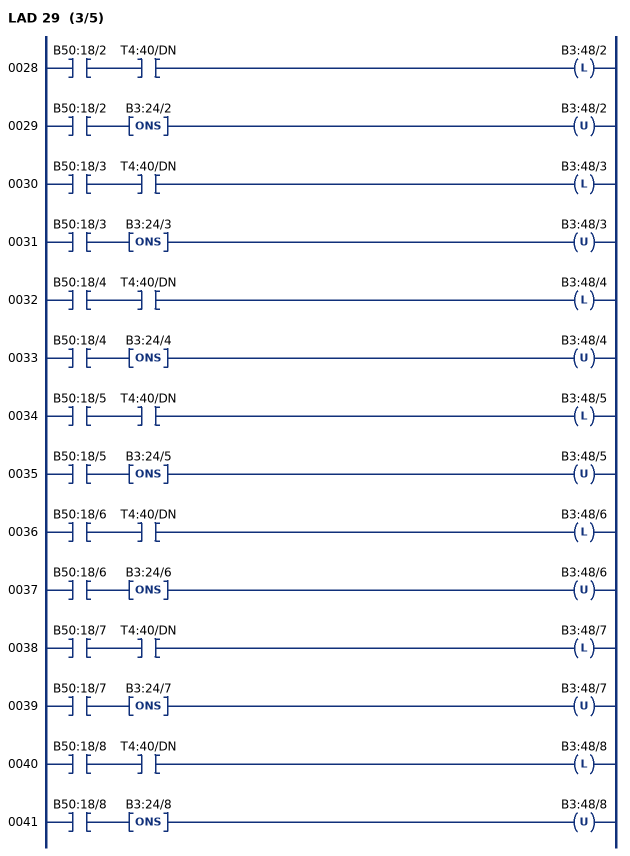
% Rung: 28 %
SOR XIC B50:18/2 XIC T4:40/DN OTL B3:48/2 EOR
% Rung: 29 %
SOR XIC B50:18/2 OSR B3:24/2 OTU B3:48/2 EOR
% Rung: 30 %
SOR XIC B50:18/3 XIC T4:40/DN OTL B3:48/3 EOR
% Rung: 31 %
SOR XIC B50:18/3 OSR B3:24/3 OTU B3:48/3 EOR
% Rung: 32 %
SOR XIC B50:18/4 XIC T4:40/DN OTL B3:48/4 EOR
% Rung: 33 %
SOR XIC B50:18/4 OSR B3:24/4 OTU B3:48/4 EOR
% Rung: 34 %
SOR XIC B50:18/5 XIC T4:40/DN OTL B3:48/5 EOR
% Rung: 35 %
SOR XIC B50:18/5 OSR B3:24/5 OTU B3:48/5 EOR
% Rung: 36 %
SOR XIC B50:18/6 XIC T4:40/DN OTL B3:48/6 EOR
% Rung: 37 %
SOR XIC B50:18/6 OSR B3:24/6 OTU B3:48/6 EOR
% Rung: 38 %
SOR XIC B50:18/7 XIC T4:40/DN OTL B3:48/7 EOR
% Rung: 39 %
SOR XIC B50:18/7 OSR B3:24/7 OTU B3:48/7 EOR
% Rung: 40 %
SOR XIC B50:18/8 XIC T4:40/DN OTL B3:48/8 EOR
% Rung: 41 %
SOR XIC B50:18/8 OSR B3:24/8 OTU B3:48/8 EOR

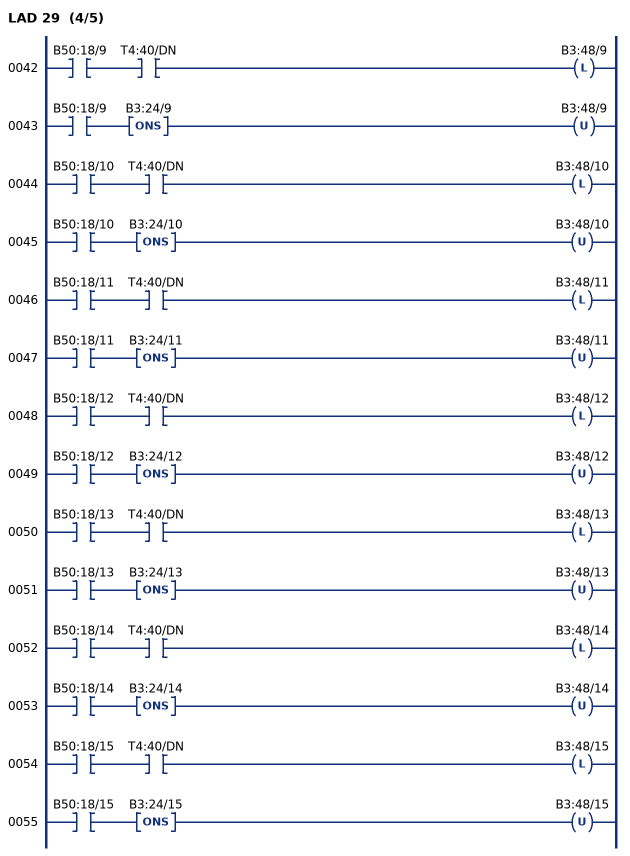
% Rung: 42 %
SOR XIC B50:18/9 XIC T4:40/DN OTL B3:48/9 EOR
% Rung: 43 %
SOR XIC B50:18/9 OSR B3:24/9 OTU B3:48/9 EOR
% Rung: 44 %
SOR XIC B50:18/10 XIC T4:40/DN OTL B3:48/10 EOR
% Rung: 45 %
SOR XIC B50:18/10 OSR B3:24/10 OTU B3:48/10 EOR
% Rung: 46 %
SOR XIC B50:18/11 XIC T4:40/DN OTL B3:48/11 EOR
% Rung: 47 %
SOR XIC B50:18/11 OSR B3:24/11 OTU B3:48/11 EOR
% Rung: 48 %
SOR XIC B50:18/12 XIC T4:40/DN OTL B3:48/12 EOR
% Rung: 49 %
SOR XIC B50:18/12 OSR B3:24/12 OTU B3:48/12 EOR
% Rung: 50 %
SOR XIC B50:18/13 XIC T4:40/DN OTL B3:48/13 EOR
% Rung: 51 %
SOR XIC B50:18/13 OSR B3:24/13 OTU B3:48/13 EOR
% Rung: 52 %
SOR XIC B50:18/14 XIC T4:40/DN OTL B3:48/14 EOR
% Rung: 53 %
SOR XIC B50:18/14 OSR B3:24/14 OTU B3:48/14 EOR
% Rung: 54 %
SOR XIC B50:18/15 XIC T4:40/DN OTL B3:48/15 EOR
% Rung: 55 %
SOR XIC B50:18/15 OSR B3:24/15 OTU B3:48/15 EOR

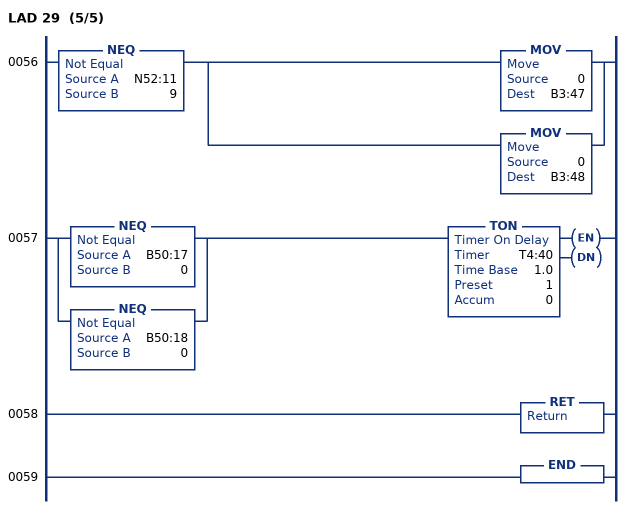
% Rung: 56 %
SOR NEQ N52:11 9 BST MOV 0 B3:47 NXB MOV 0 B3:48 BND EOR
% Rung: 57 %
SOR BST NEQ B50:17 0 NXB NEQ B50:18 0 BND TON T4:40 1.0 1 0 EOR
% Rung: 58 %
SOR RET EOR
% Rung: 59 %
SOR END EOR

LADDER 30
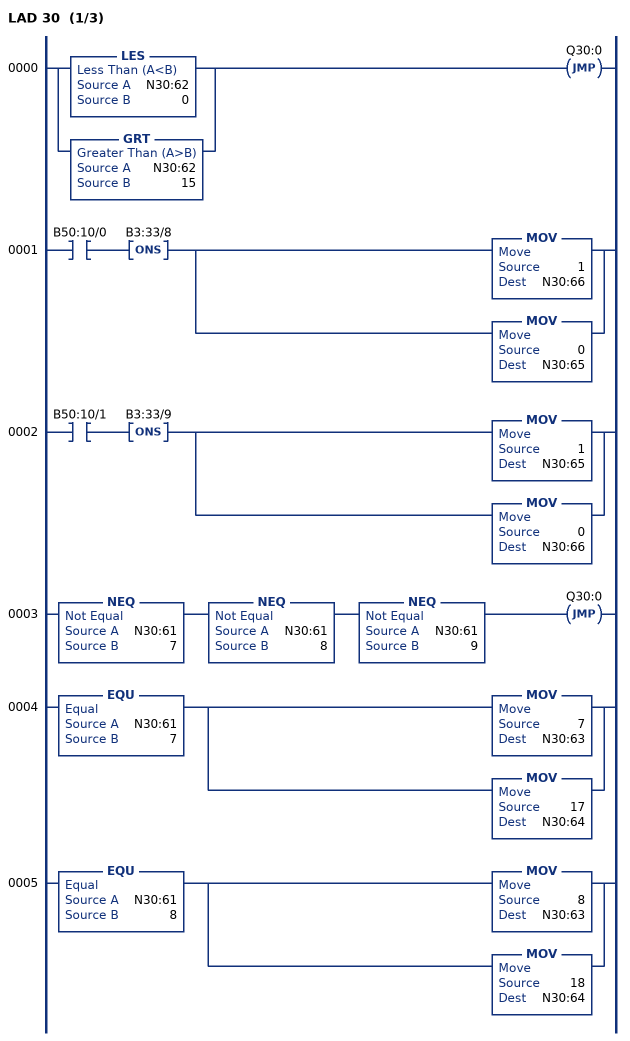
% Rung: 0 %
SOR BST LES N30:62 0 NXB GRT N30:62 15 BND JMP Q30:0 EOR
% Rung: 1 %
SOR XIC B50:10/0 OSR B3:33/8 BST MOV 1 N30:66 NXB MOV 0 N30:65 BND EOR
% Rung: 2 %
SOR XIC B50:10/1 OSR B3:33/9 BST MOV 1 N30:65 NXB MOV 0 N30:66 BND EOR
% Rung: 3 %
SOR NEQ N30:61 7 NEQ N30:61 8 NEQ N30:61 9 JMP Q30:0 EOR
% Rung: 4 %
SOR EQU N30:61 7 BST MOV 7 N30:63 NXB MOV 17 N30:64 BND EOR
% Rung: 5 %
SOR EQU N30:61 8 BST MOV 8 N30:63 NXB MOV 18 N30:64 BND EOR

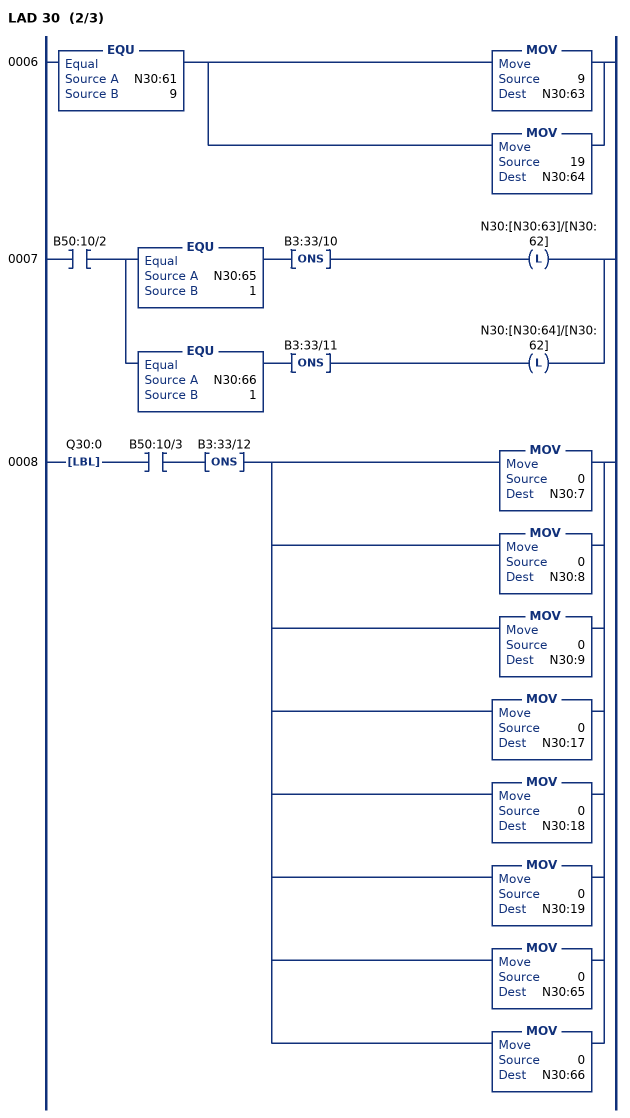
% Rung: 6 %
SOR EQU N30:61 9 BST MOV 9 N30:63 NXB MOV 19 N30:64 BND EOR
% Rung: 7 %
SOR XIC B50:10/2 BST EQU N30:65 1 OSR B3:33/10 OTL N30:[N30:63]/[N30:62] NXB EQU N30:66 1 OSR B3:33/11 OTL N30:[N30:64]/[N30:62] BND EOR
% Rung: 8 %
SOR LBL Q30:0 XIC B50:10/3 OSR B3:33/12 BST MOV 0 N30:7 NXB MOV 0 N30:8 NXB MOV 0 N30:9 NXB MOV 0 N30:17 NXB MOV 0 N30:18 NXB MOV 0 N30:19 NXB MOV 0 N30:65 NXB MOV 0 N30:66 BND EOR

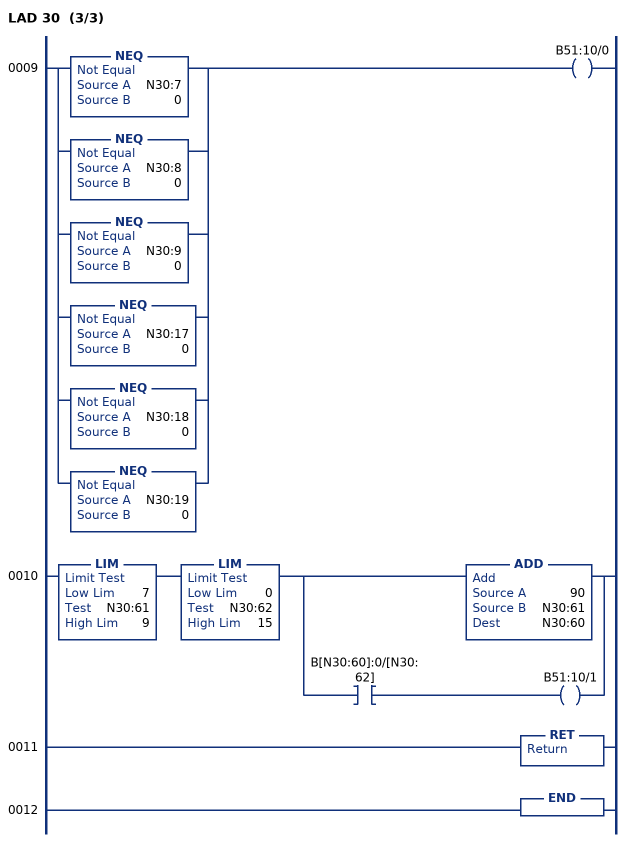
% Rung: 9 %
SOR BST NEQ N30:7 0 NXB NEQ N30:8 0 NXB NEQ N30:9 0 NXB NEQ N30:17 0 NXB NEQ N30:18 0 NXB NEQ N30:19 0 BND OTE B51:10/0 EOR
% Rung: 10 %
SOR LIM 7 N30:61 9 LIM 0 N30:62 15 BST ADD 90 N30:61 N30:60 NXB XIC B[N30:60]:0/[N30:62] OTE B51:10/1 BND EOR
% Rung: 11 %
SOR RET EOR
% Rung: 12 %
SOR END EOR

LADDER 31
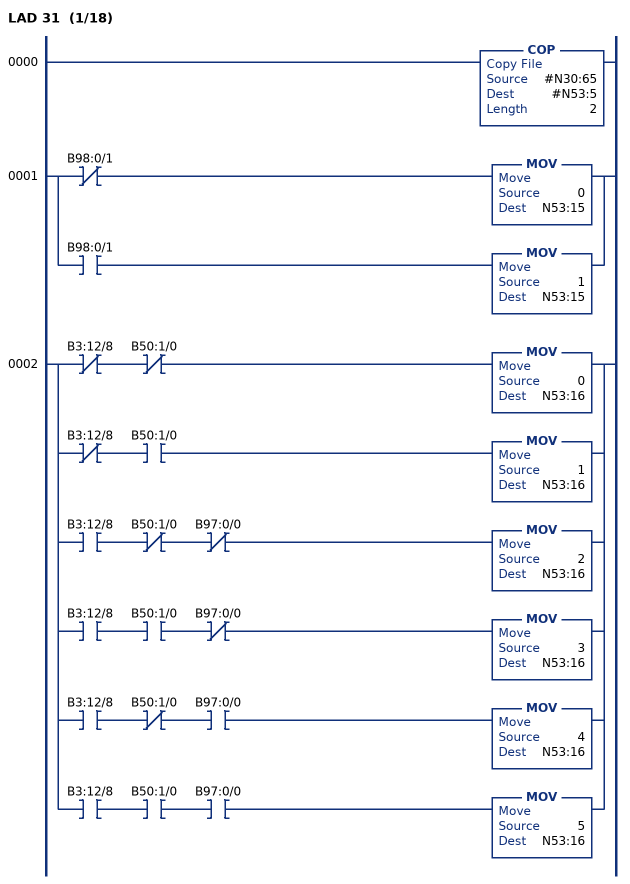
% Rung: 0 %
SOR COP #N30:65 #N53:5 2 EOR
% Rung: 1 %
SOR BST XIO B98:0/1 MOV 0 N53:15 NXB XIC B98:0/1 MOV 1 N53:15 BND EOR
% Rung: 2 %
SOR BST XIO B3:12/8 XIO B50:1/0 MOV 0 N53:16 NXB XIO B3:12/8 XIC B50:1/0 MOV 1 N53:16 NXB XIC B3:12/8 XIO B50:1/0 XIO B97:0/0 MOV 2 N53:16 NXB XIC B3:12/8 XIC B50:1/0 XIO B97:0/0 MOV 3 N53:16 NXB XIC B3:12/8 XIO B50:1/0 XIC B97:0/0 MOV 4 N53:16 NXB XIC B3:12/8 XIC B50:1/0 XIC B97:0/0 MOV 5 N53:16 BND EOR

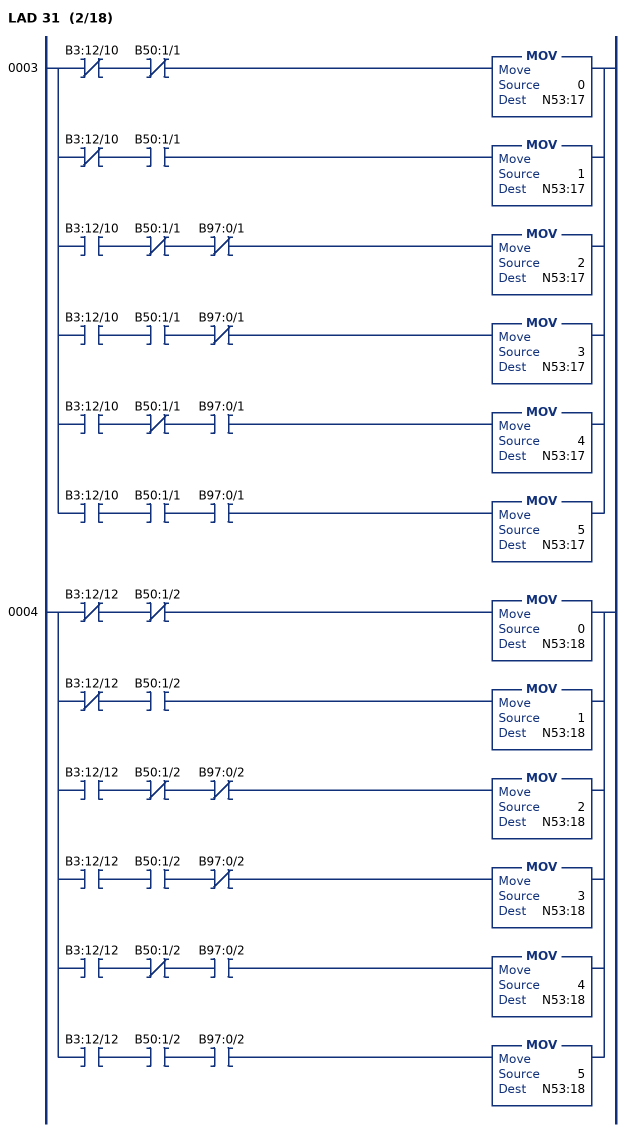
% Rung: 3 %
SOR BST XIO B3:12/10 XIO B50:1/1 MOV 0 N53:17 NXB XIO B3:12/10 XIC B50:1/1 MOV 1 N53:17 NXB XIC B3:12/10 XIO B50:1/1 XIO B97:0/1 MOV 2 N53:17 NXB XIC B3:12/10 XIC B50:1/1 XIO B97:0/1 MOV 3 N53:17 NXB XIC B3:12/10 XIO B50:1/1 XIC B97:0/1 MOV 4 N53:17 NXB XIC B3:12/10 XIC B50:1/1 XIC B97:0/1 MOV 5 N53:17 BND EOR
% Rung: 4 %
SOR BST XIO B3:12/12 XIO B50:1/2 MOV 0 N53:18 NXB XIO B3:12/12 XIC B50:1/2 MOV 1 N53:18 NXB XIC B3:12/12 XIO B50:1/2 XIO B97:0/2 MOV 2 N53:18 NXB XIC B3:12/12 XIC B50:1/2 XIO B97:0/2 MOV 3 N53:18 NXB XIC B3:12/12 XIO B50:1/2 XIC B97:0/2 MOV 4 N53:18 NXB XIC B3:12/12 XIC B50:1/2 XIC B97:0/2 MOV 5 N53:18 BND EOR

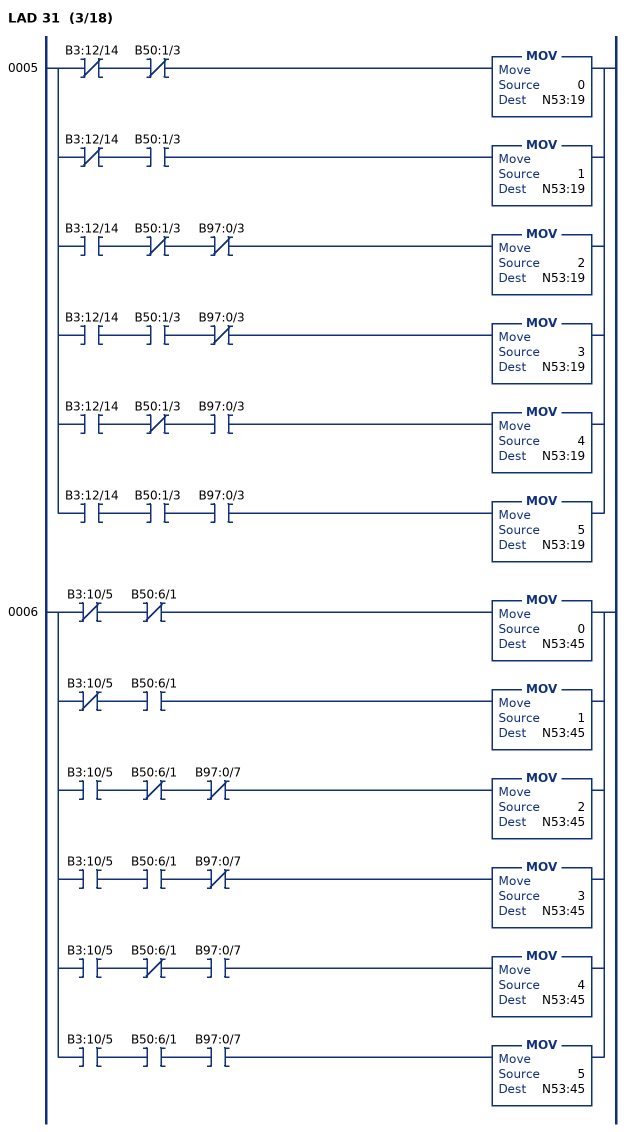
% Rung: 5 %
SOR BST XIO B3:12/14 XIO B50:1/3 MOV 0 N53:19 NXB XIO B3:12/14 XIC B50:1/3 MOV 1 N53:19 NXB XIC B3:12/14 XIO B50:1/3 XIO B97:0/3 MOV 2 N53:19 NXB XIC B3:12/14 XIC B50:1/3 XIO B97:0/3 MOV 3 N53:19 NXB XIC B3:12/14 XIO B50:1/3 XIC B97:0/3 MOV 4 N53:19 NXB XIC B3:12/14 XIC B50:1/3 XIC B97:0/3 MOV 5 N53:19 BND EOR
% Rung: 6 %
SOR BST XIO B3:10/5 XIO B50:6/1 MOV 0 N53:45 NXB XIO B3:10/5 XIC B50:6/1 MOV 1 N53:45 NXB XIC B3:10/5 XIO B50:6/1 XIO B97:0/7 MOV 2 N53:45 NXB XIC B3:10/5 XIC B50:6/1 XIO B97:0/7 MOV 3 N53:45 NXB XIC B3:10/5 XIO B50:6/1 XIC B97:0/7 MOV 4 N53:45 NXB XIC B3:10/5 XIC B50:6/1 XIC B97:0/7 MOV 5 N53:45 BND EOR

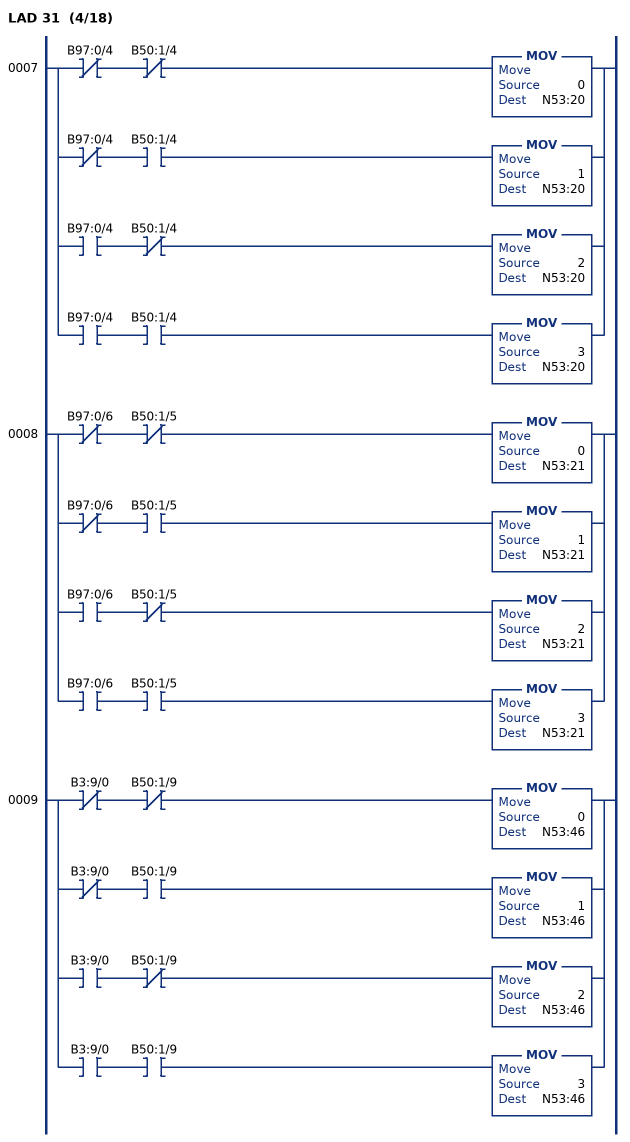
% Rung: 7 %
SOR BST XIO B97:0/4 XIO B50:1/4 MOV 0 N53:20 NXB XIO B97:0/4 XIC B50:1/4 MOV 1 N53:20 NXB XIC B97:0/4 XIO B50:1/4 MOV 2 N53:20 NXB XIC B97:0/4 XIC B50:1/4 MOV 3 N53:20 BND EOR
% Rung: 8 %
SOR BST XIO B97:0/6 XIO B50:1/5 MOV 0 N53:21 NXB XIO B97:0/6 XIC B50:1/5 MOV 1 N53:21 NXB XIC B97:0/6 XIO B50:1/5 MOV 2 N53:21 NXB XIC B97:0/6 XIC B50:1/5 MOV 3 N53:21 BND EOR
% Rung: 9 %
SOR BST XIO B3:9/0 XIO B50:1/9 MOV 0 N53:46 NXB XIO B3:9/0 XIC B50:1/9 MOV 1 N53:46 NXB XIC B3:9/0 XIO B50:1/9 MOV 2 N53:46 NXB XIC B3:9/0 XIC B50:1/9 MOV 3 N53:46 BND EOR

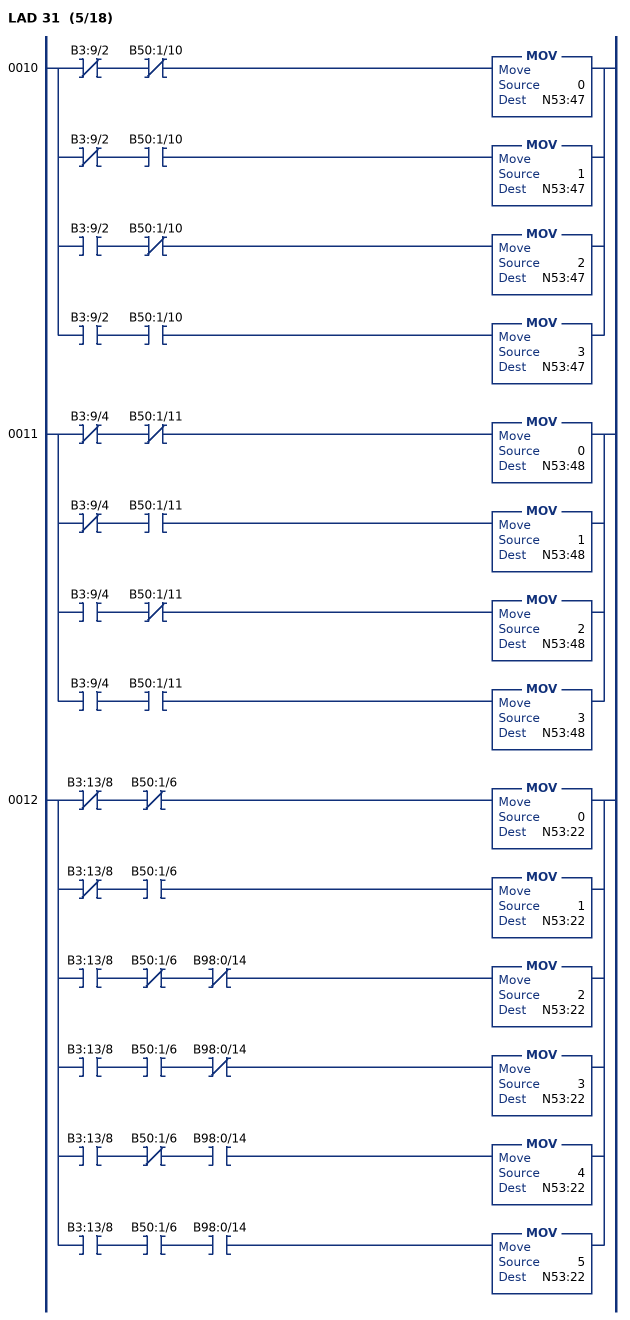
% Rung: 10 %
SOR BST XIO B3:9/2 XIO B50:1/10 MOV 0 N53:47 NXB XIO B3:9/2 XIC B50:1/10 MOV 1 N53:47 NXB XIC B3:9/2 XIO B50:1/10 MOV 2 N53:47 NXB XIC B3:9/2 XIC B50:1/10 MOV 3 N53:47 BND EOR
% Rung: 11 %
SOR BST XIO B3:9/4 XIO B50:1/11 MOV 0 N53:48 NXB XIO B3:9/4 XIC B50:1/11 MOV 1 N53:48 NXB XIC B3:9/4 XIO B50:1/11 MOV 2 N53:48 NXB XIC B3:9/4 XIC B50:1/11 MOV 3 N53:48 BND EOR
% Rung: 12 %
SOR BST XIO B3:13/8 XIO B50:1/6 MOV 0 N53:22 NXB XIO B3:13/8 XIC B50:1/6 MOV 1 N53:22 NXB XIC B3:13/8 XIO B50:1/6 XIO B98:0/14 MOV 2 N53:22 NXB XIC B3:13/8 XIC B50:1/6 XIO B98:0/14 MOV 3 N53:22 NXB XIC B3:13/8 XIO B50:1/6 XIC B98:0/14 MOV 4 N53:22 NXB XIC B3:13/8 XIC B50:1/6 XIC B98:0/14 MOV 5 N53:22 BND EOR

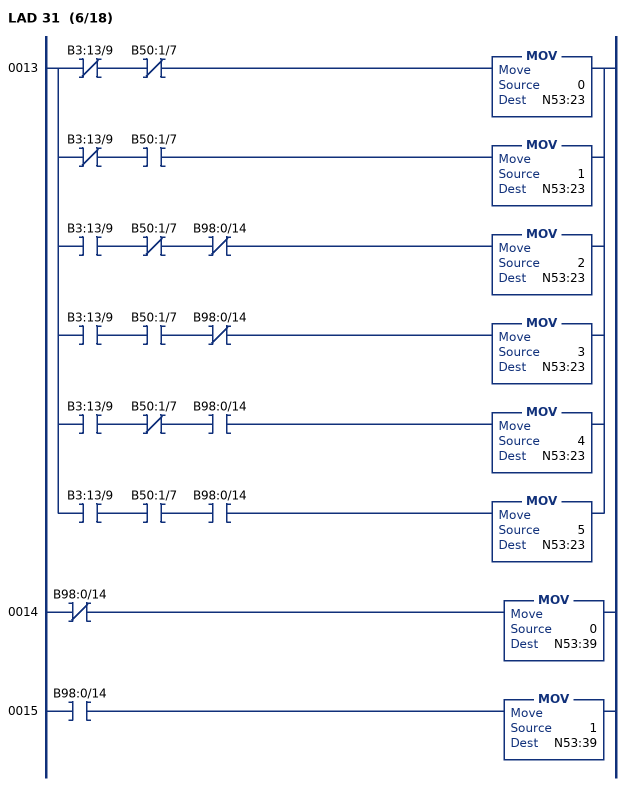
% Rung: 13 %
SOR BST XIO B3:13/9 XIO B50:1/7 MOV 0 N53:23 NXB XIO B3:13/9 XIC B50:1/7 MOV 1 N53:23 NXB XIC B3:13/9 XIO B50:1/7 XIO B98:0/14 MOV 2 N53:23 NXB XIC B3:13/9 XIC B50:1/7 XIO B98:0/14 MOV 3 N53:23 NXB XIC B3:13/9 XIO B50:1/7 XIC B98:0/14 MOV 4 N53:23 NXB XIC B3:13/9 XIC B50:1/7 XIC B98:0/14 MOV 5 N53:23 BND EOR
% Rung: 14 %
SOR XIO B98:0/14 MOV 0 N53:39 EOR
% Rung: 15 %
SOR XIC B98:0/14 MOV 1 N53:39 EOR

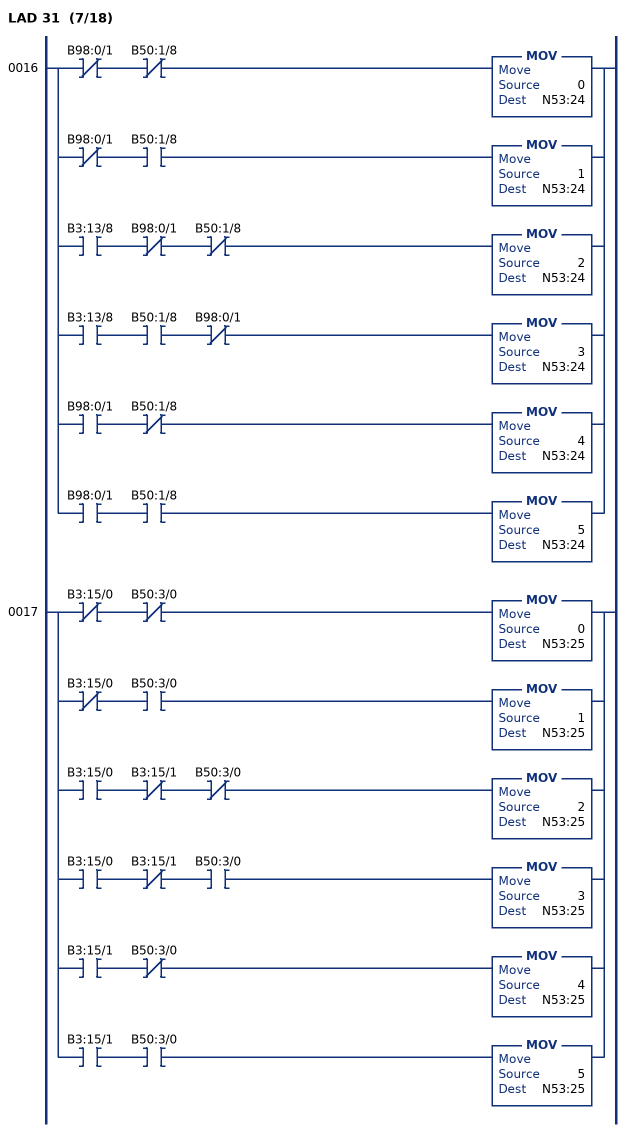
% Rung: 16 %
SOR BST XIO B98:0/1 XIO B50:1/8 MOV 0 N53:24 NXB XIO B98:0/1 XIC B50:1/8 MOV 1 N53:24 NXB XIC B3:13/8 XIO B98:0/1 XIO B50:1/8 MOV 2 N53:24 NXB XIC B3:13/8 XIC B50:1/8 XIO B98:0/1 MOV 3 N53:24 NXB XIC B98:0/1 XIO B50:1/8 MOV 4 N53:24 NXB XIC B98:0/1 XIC B50:1/8 MOV 5 N53:24 BND EOR
% Rung: 17 %
SOR BST XIO B3:15/0 XIO B50:3/0 MOV 0 N53:25 NXB XIO B3:15/0 XIC B50:3/0 MOV 1 N53:25 NXB XIC B3:15/0 XIO B3:15/1 XIO B50:3/0 MOV 2 N53:25 NXB XIC B3:15/0 XIO B3:15/1 XIC B50:3/0 MOV 3 N53:25 NXB XIC B3:15/1 XIO B50:3/0 MOV 4 N53:25 NXB XIC B3:15/1 XIC B50:3/0 MOV 5 N53:25 BND EOR

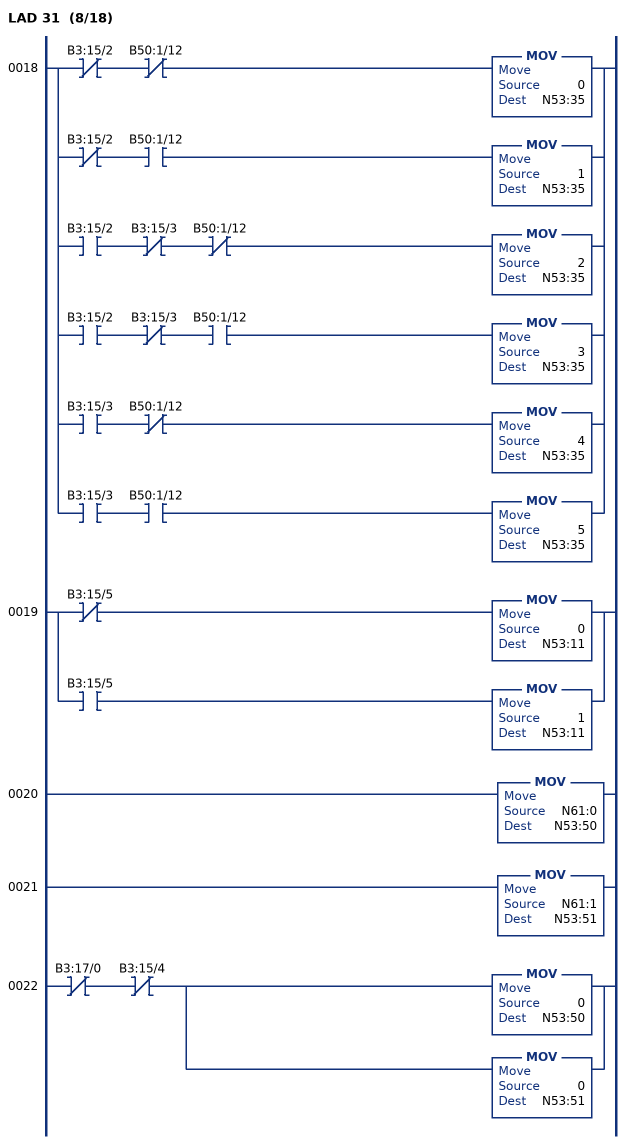
% Rung: 18 %
SOR BST XIO B3:15/2 XIO B50:1/12 MOV 0 N53:35 NXB XIO B3:15/2 XIC B50:1/12 MOV 1 N53:35 NXB XIC B3:15/2 XIO B3:15/3 XIO B50:1/12 MOV 2 N53:35 NXB XIC B3:15/2 XIO B3:15/3 XIC B50:1/12 MOV 3 N53:35 NXB XIC B3:15/3 XIO B50:1/12 MOV 4 N53:35 NXB XIC B3:15/3 XIC B50:1/12 MOV 5 N53:35 BND EOR
% Rung: 19 %
SOR BST XIO B3:15/5 MOV 0 N53:11 NXB XIC B3:15/5 MOV 1 N53:11 BND EOR
% Rung: 20 %
SOR MOV N61:0 N53:50 EOR
% Rung: 21 %
SOR MOV N61:1 N53:51 EOR
% Rung: 22 %
SOR XIO B3:17/0 XIO B3:15/4 BST MOV 0 N53:50 NXB MOV 0 N53:51 BND EOR

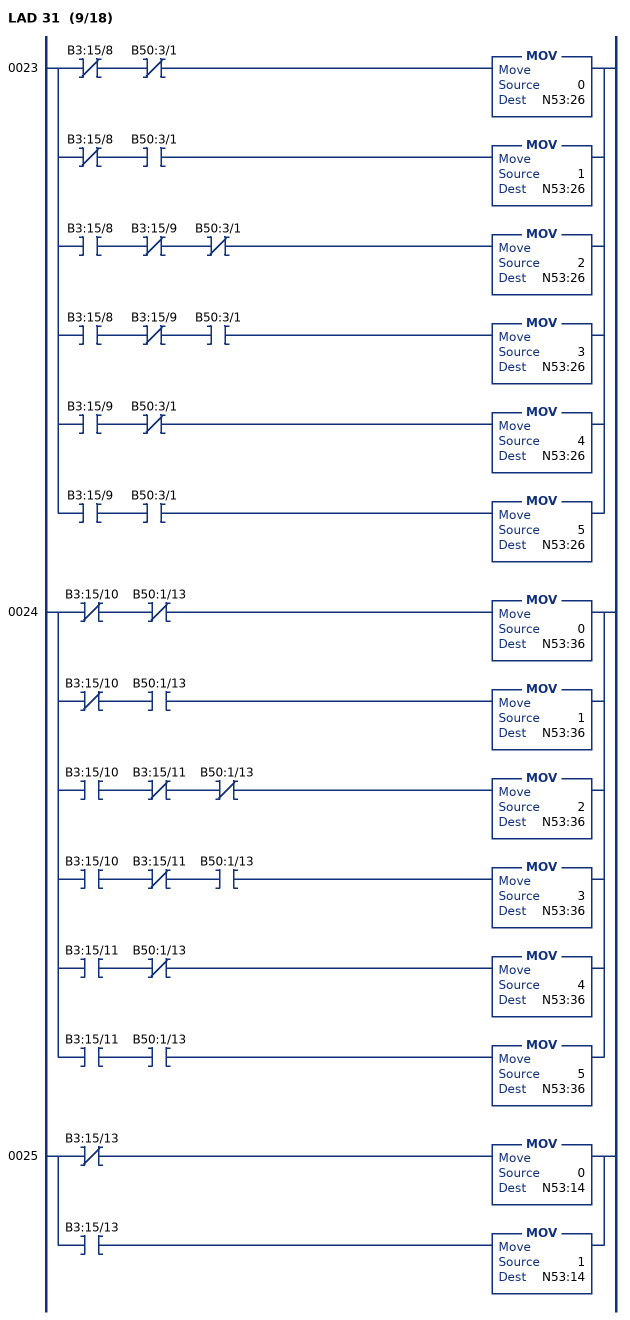
% Rung: 23 %
SOR BST XIO B3:15/8 XIO B50:3/1 MOV 0 N53:26 NXB XIO B3:15/8 XIC B50:3/1 MOV 1 N53:26 NXB XIC B3:15/8 XIO B3:15/9 XIO B50:3/1 MOV 2 N53:26 NXB XIC B3:15/8 XIO B3:15/9 XIC B50:3/1 MOV 3 N53:26 NXB XIC B3:15/9 XIO B50:3/1 MOV 4 N53:26 NXB XIC B3:15/9 XIC B50:3/1 MOV 5 N53:26 BND EOR
% Rung: 24 %
SOR BST XIO B3:15/10 XIO B50:1/13 MOV 0 N53:36 NXB XIO B3:15/10 XIC B50:1/13 MOV 1 N53:36 NXB XIC B3:15/10 XIO B3:15/11 XIO B50:1/13 MOV 2 N53:36 NXB XIC B3:15/10 XIO B3:15/11 XIC B50:1/13 MOV 3 N53:36 NXB XIC B3:15/11 XIO B50:1/13 MOV 4 N53:36 NXB XIC B3:15/11 XIC B50:1/13 MOV 5 N53:36 BND EOR
% Rung: 25 %
SOR BST XIO B3:15/13 MOV 0 N53:14 NXB XIC B3:15/13 MOV 1 N53:14 BND EOR

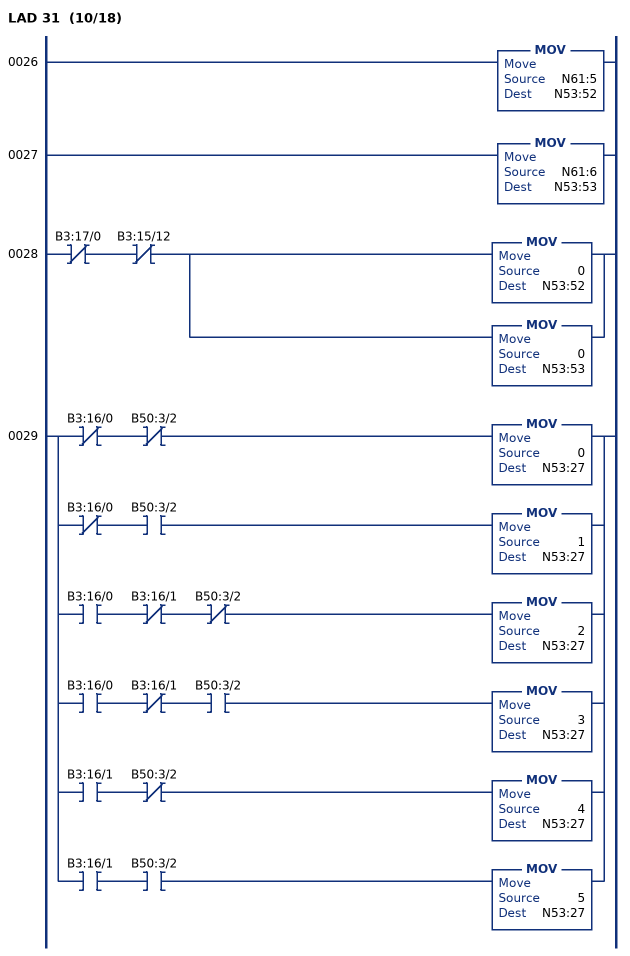
% Rung: 26 %
SOR MOV N61:5 N53:52 EOR
% Rung: 27 %
SOR MOV N61:6 N53:53 EOR
% Rung: 28 %
SOR XIO B3:17/0 XIO B3:15/12 BST MOV 0 N53:52 NXB MOV 0 N53:53 BND EOR
% Rung: 29 %
SOR BST XIO B3:16/0 XIO B50:3/2 MOV 0 N53:27 NXB XIO B3:16/0 XIC B50:3/2 MOV 1 N53:27 NXB XIC B3:16/0 XIO B3:16/1 XIO B50:3/2 MOV 2 N53:27 NXB XIC B3:16/0 XIO B3:16/1 XIC B50:3/2 MOV 3 N53:27 NXB XIC B3:16/1 XIO B50:3/2 MOV 4 N53:27 NXB XIC B3:16/1 XIC B50:3/2 MOV 5 N53:27 BND EOR

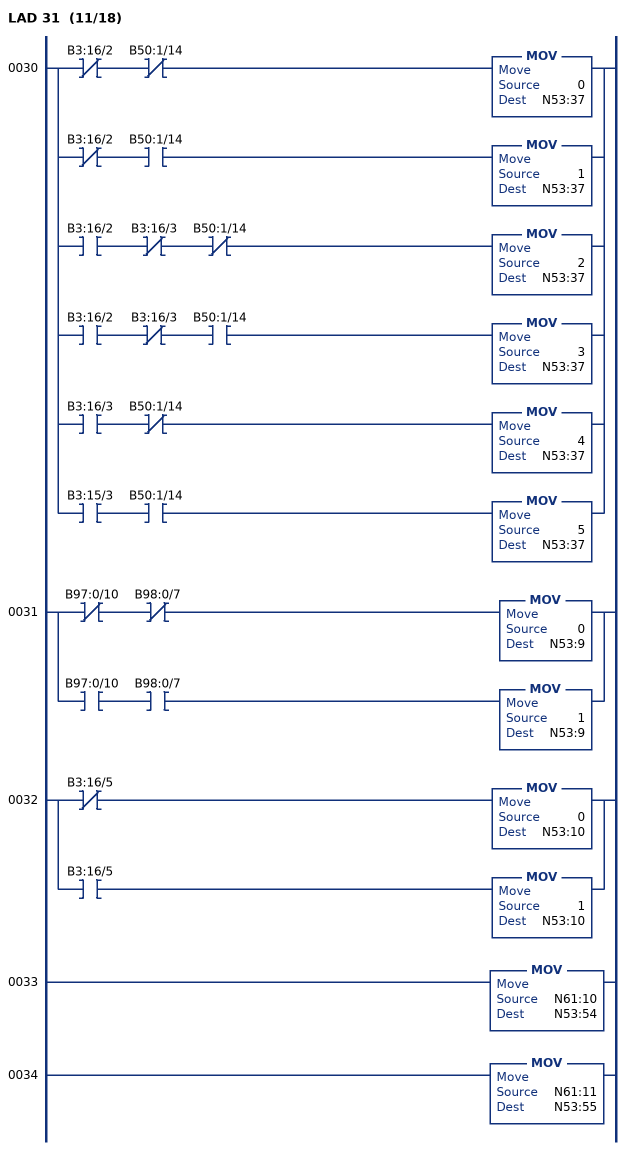
% Rung: 30 %
SOR BST XIO B3:16/2 XIO B50:1/14 MOV 0 N53:37 NXB XIO B3:16/2 XIC B50:1/14 MOV 1 N53:37 NXB XIC B3:16/2 XIO B3:16/3 XIO B50:1/14 MOV 2 N53:37 NXB XIC B3:16/2 XIO B3:16/3 XIC B50:1/14 MOV 3 N53:37 NXB XIC B3:16/3 XIO B50:1/14 MOV 4 N53:37 NXB XIC B3:15/3 XIC B50:1/14 MOV 5 N53:37 BND EOR
% Rung: 31 %
SOR BST XIO B97:0/10 XIO B98:0/7 MOV 0 N53:9 NXB XIC B97:0/10 XIC B98:0/7 MOV 1 N53:9 BND EOR
% Rung: 32 %
SOR BST XIO B3:16/5 MOV 0 N53:10 NXB XIC B3:16/5 MOV 1 N53:10 BND EOR
% Rung: 33 %
SOR MOV N61:10 N53:54 EOR
% Rung: 34 %
SOR MOV N61:11 N53:55 EOR

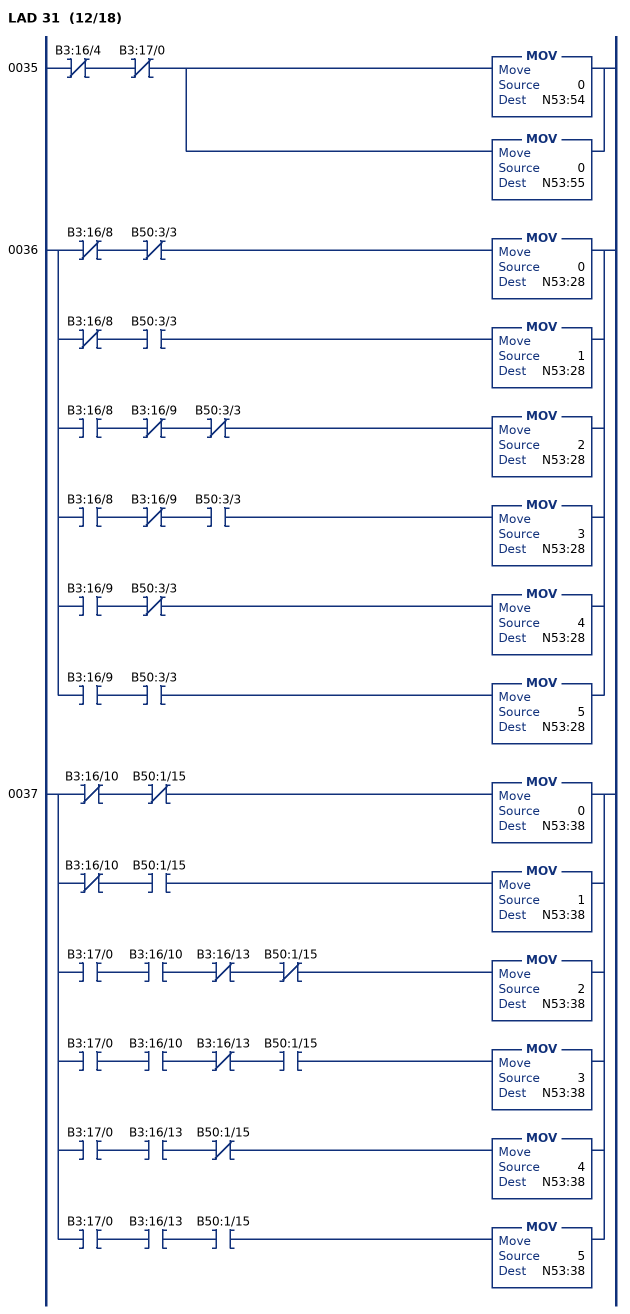
% Rung: 35 %
SOR XIO B3:16/4 XIO B3:17/0 BST MOV 0 N53:54 NXB MOV 0 N53:55 BND EOR
% Rung: 36 %
SOR BST XIO B3:16/8 XIO B50:3/3 MOV 0 N53:28 NXB XIO B3:16/8 XIC B50:3/3 MOV 1 N53:28 NXB XIC B3:16/8 XIO B3:16/9 XIO B50:3/3 MOV 2 N53:28 NXB XIC B3:16/8 XIO B3:16/9 XIC B50:3/3 MOV 3 N53:28 NXB XIC B3:16/9 XIO B50:3/3 MOV 4 N53:28 NXB XIC B3:16/9 XIC B50:3/3 MOV 5 N53:28 BND EOR
% Rung: 37 %
SOR BST XIO B3:16/10 XIO B50:1/15 MOV 0 N53:38 NXB XIO B3:16/10 XIC B50:1/15 MOV 1 N53:38 NXB XIC B3:17/0 XIC B3:16/10 XIO B3:16/13 XIO B50:1/15 MOV 2 N53:38 NXB XIC B3:17/0 XIC B3:16/10 XIO B3:16/13 XIC B50:1/15 MOV 3 N53:38 NXB XIC B3:17/0 XIC B3:16/13 XIO B50:1/15 MOV 4 N53:38 NXB XIC B3:17/0 XIC B3:16/13 XIC B50:1/15 MOV 5 N53:38 BND EOR

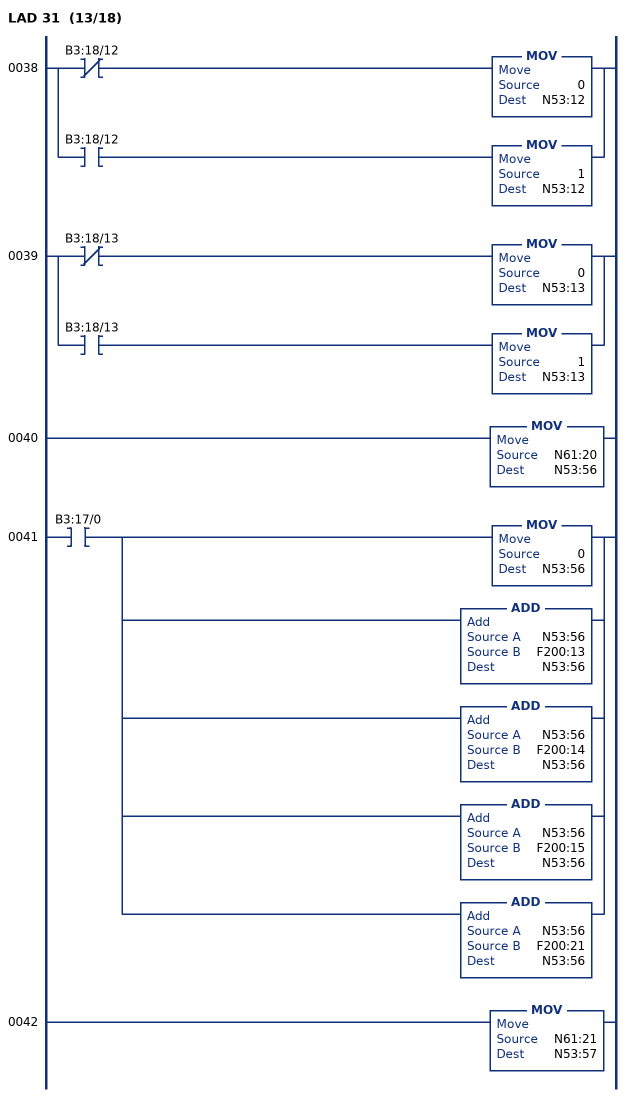
% Rung: 38 %
SOR BST XIO B3:18/12 MOV 0 N53:12 NXB XIC B3:18/12 MOV 1 N53:12 BND EOR
% Rung: 39 %
SOR BST XIO B3:18/13 MOV 0 N53:13 NXB XIC B3:18/13 MOV 1 N53:13 BND EOR
% Rung: 40 %
SOR MOV N61:20 N53:56 EOR
% Rung: 41 %
SOR XIC B3:17/0 BST MOV 0 N53:56 NXB ADD N53:56 F200:13 N53:56 NXB ADD N53:56 F200:14 N53:56 NXB ADD N53:56 F200:15 N53:56 NXB ADD N53:56 F200:21 N53:56 BND EOR
% Rung: 42 %
SOR MOV N61:21 N53:57 EOR

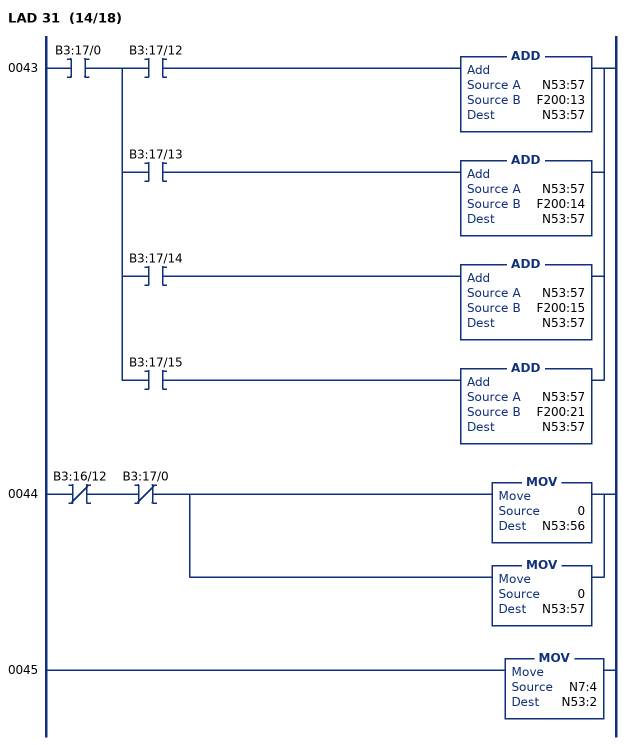
% Rung: 43 %
SOR XIC B3:17/0 BST XIC B3:17/12 ADD N53:57 F200:13 N53:57 NXB XIC B3:17/13 ADD N53:57 F200:14 N53:57 NXB XIC B3:17/14 ADD N53:57 F200:15 N53:57 NXB XIC B3:17/15 ADD N53:57 F200:21 N53:57 BND EOR
% Rung: 44 %
SOR XIO B3:16/12 XIO B3:17/0 BST MOV 0 N53:56 NXB MOV 0 N53:57 BND EOR
% Rung: 45 %
SOR MOV N7:4 N53:2 EOR

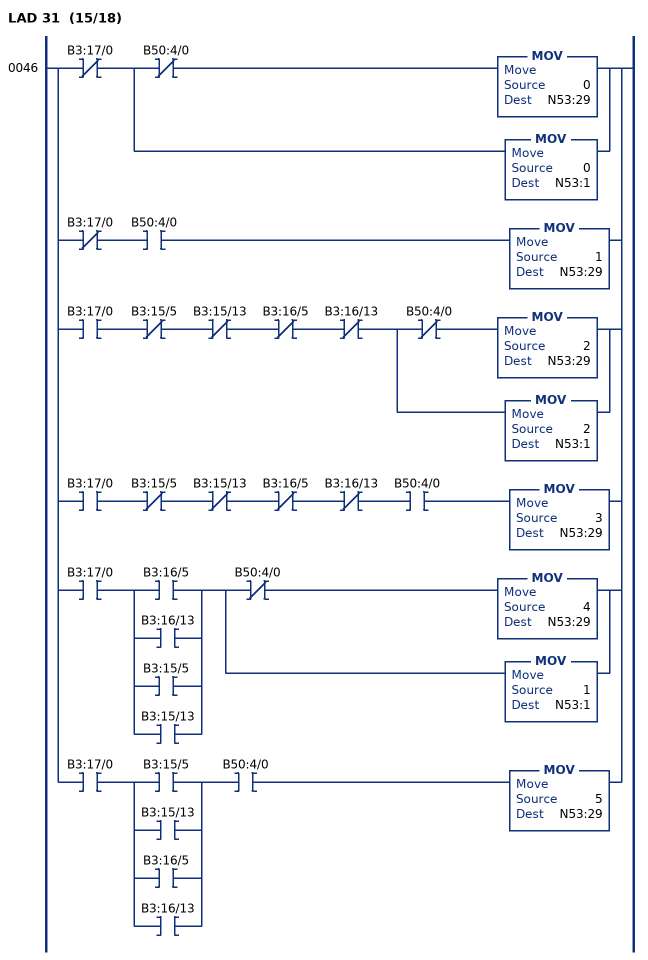
% Rung: 46 %
SOR BST XIO B3:17/0 BST XIO B50:4/0 MOV 0 N53:29 NXB MOV 0 N53:1 BND NXB XIO B3:17/0 XIC B50:4/0 MOV 1 N53:29 NXB XIC B3:17/0 XIO B3:15/5 XIO B3:15/13 XIO B3:16/5 XIO B3:16/13 BST XIO B50:4/0 MOV 2 N53:29 NXB MOV 2 N53:1 BND NXB XIC B3:17/0 XIO B3:15/5 XIO B3:15/13 XIO B3:16/5 XIO B3:16/13 XIC B50:4/0 MOV 3 N53:29 NXB XIC B3:17/0 BST XIC B3:16/5 NXB XIC B3:16/13 NXB XIC B3:15/5 NXB XIC B3:15/13 BND BST XIO B50:4/0 MOV 4 N53:29 NXB MOV 1 N53:1 BND NXB XIC B3:17/0 BST XIC B3:15/5 NXB XIC B3:15/13 NXB XIC B3:16/5 NXB XIC B3:16/13 BND XIC B50:4/0 MOV 5 N53:29 BND EOR

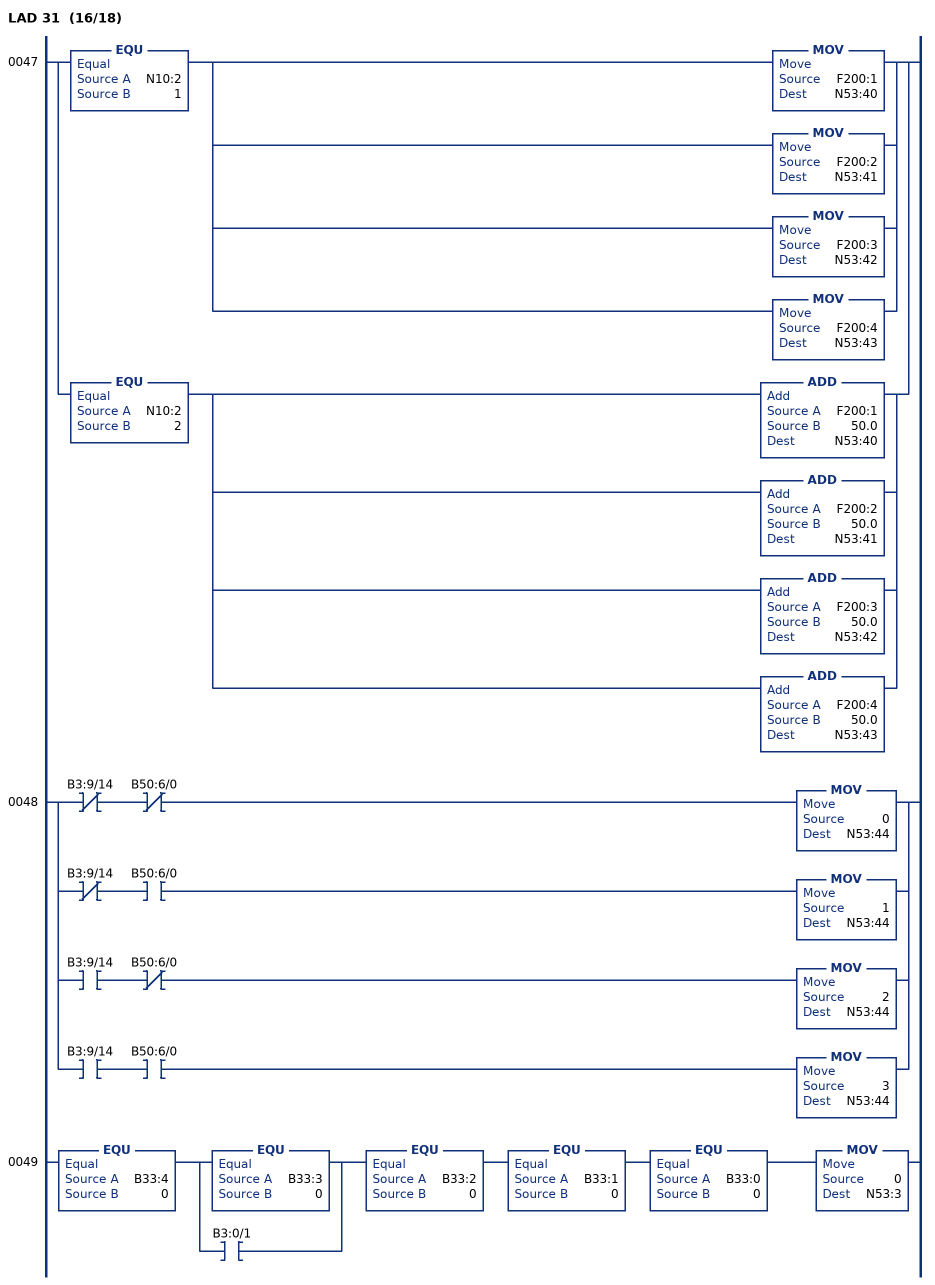
% Rung: 47 %
SOR BST EQU N10:2 1 BST MOV F200:1 N53:40 NXB MOV F200:2 N53:41 NXB MOV F200:3 N53:42 NXB MOV F200:4 N53:43 BND NXB EQU N10:2 2 BST ADD F200:1 50.0 N53:40 NXB ADD F200:2 50.0 N53:41 NXB ADD F200:3 50.0 N53:42 NXB ADD F200:4 50.0 N53:43 BND BND EOR
% Rung: 48 %
SOR BST XIO B3:9/14 XIO B50:6/0 MOV 0 N53:44 NXB XIO B3:9/14 XIC B50:6/0 MOV 1 N53:44 NXB XIC B3:9/14 XIO B50:6/0 MOV 2 N53:44 NXB XIC B3:9/14 XIC B50:6/0 MOV 3 N53:44 BND EOR
% Rung: 49 %
SOR EQU B33:4 0 BST EQU B33:3 0 NXB XIC B3:0/1 BND EQU B33:2 0 EQU B33:1 0 EQU B33:0 0 MOV 0 N53:3 EOR

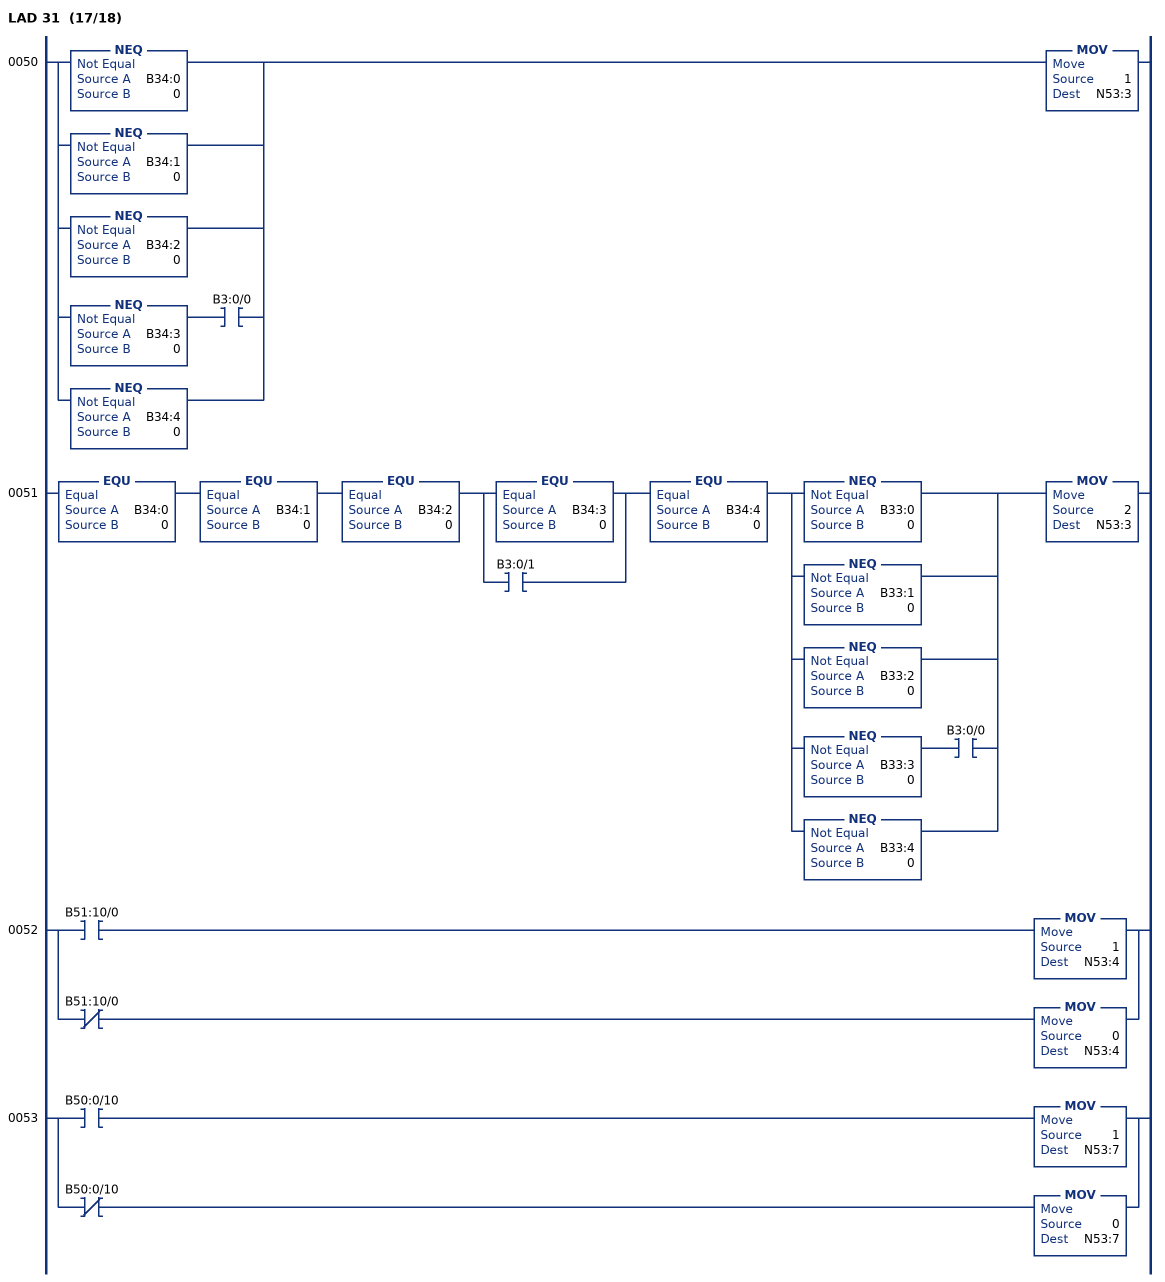
% Rung: 50 %
SOR BST NEQ B34:0 0 NXB NEQ B34:1 0 NXB NEQ B34:2 0 NXB NEQ B34:3 0 XIC B3:0/0 NXB NEQ B34:4 0 BND MOV 1 N53:3 EOR
% Rung: 51 %
SOR EQU B34:0 0 EQU B34:1 0 EQU B34:2 0 BST EQU B34:3 0 NXB XIC B3:0/1 BND EQU B34:4 0 BST NEQ B33:0 0 NXB NEQ B33:1 0 NXB NEQ B33:2 0 NXB NEQ B33:3 0 XIC B3:0/0 NXB NEQ B33:4 0 BND MOV 2 N53:3 EOR
% Rung: 52 %
SOR BST XIC B51:10/0 MOV 1 N53:4 NXB XIO B51:10/0 MOV 0 N53:4 BND EOR
% Rung: 53 %
SOR BST XIC B50:0/10 MOV 1 N53:7 NXB XIO B50:0/10 MOV 0 N53:7 BND EOR

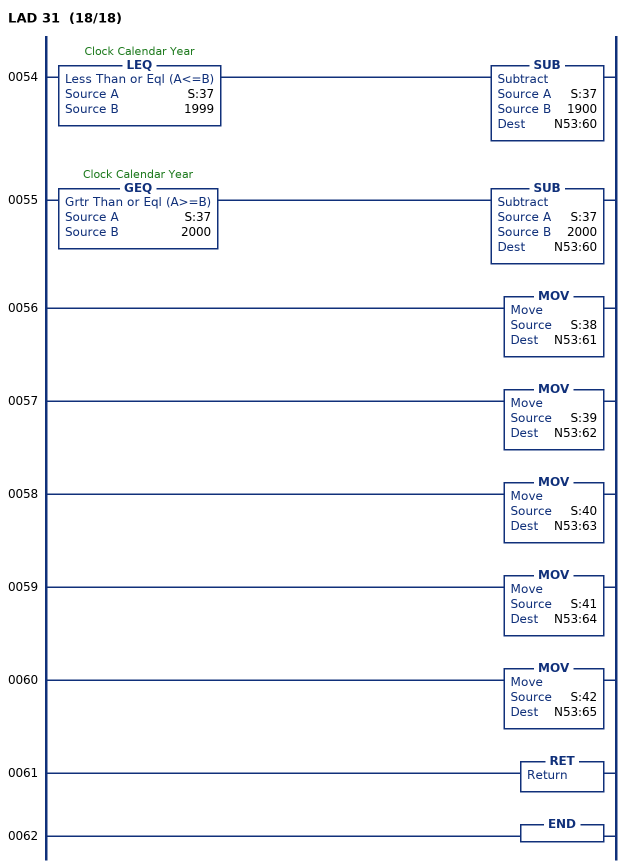
% Rung: 54 %
SOR LEQ S:37 1999 SUB S:37 1900 N53:60 EOR
%   S:37  "Clock Calendar Year" %
% Rung: 55 %
SOR GEQ S:37 2000 SUB S:37 2000 N53:60 EOR
%   S:37  "Clock Calendar Year" %
% Rung: 56 %
SOR MOV S:38 N53:61 EOR
%   S:38  "Clock Calendar Month" %
% Rung: 57 %
SOR MOV S:39 N53:62 EOR
%   S:39  "Clock Calendar Day" %
% Rung: 58 %
SOR MOV S:40 N53:63 EOR
%   S:40  "Clock Calendar Hours" %
% Rung: 59 %
SOR MOV S:41 N53:64 EOR
%   S:41  "Clock Calendar Minutes" %
% Rung: 60 %
SOR MOV S:42 N53:65 EOR
%   S:42  "Clock Calendar Seconds" %
% Rung: 61 %
SOR RET EOR
% Rung: 62 %
SOR END EOR

LADDER 32
